Staubli VAL3: clkValve5.pgx

program clkValve5()
begin
  call toggleValve(5)
end
